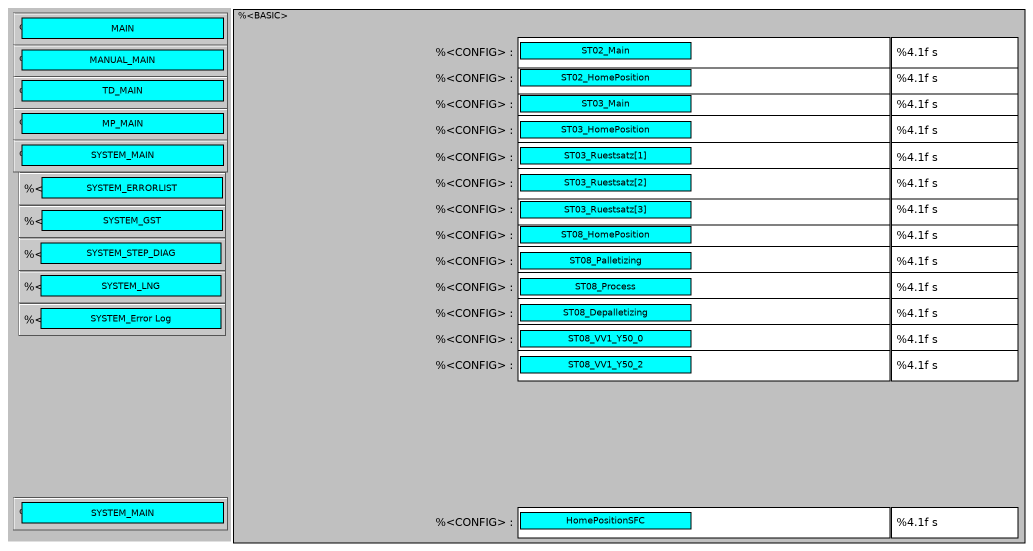
[picture p142: SYSTEM_STEP_DIAG (HMI screen)]
rectangle at (228,115)-(1020,649): text "%<BASIC>"; shows 'Prozess-Schrittketten'
embedded screen at (3,114)-(226,647): M0003_System
embedded screen at (282,195)-(1013,226): ZLIB_SFC_STATE
embedded screen at (282,221)-(1013,252): ZLIB_SFC_STATE
embedded screen at (282,326)-(1013,357): ZLIB_SFC_STATE
embedded screen at (282,352)-(1013,383): ZLIB_SFC_STATE
embedded screen at (282,378)-(1013,409): ZLIB_SFC_STATE
embedded screen at (282,404)-(1013,435): ZLIB_SFC_STATE
embedded screen at (282,430)-(1013,461): ZLIB_SFC_STATE
embedded screen at (282,456)-(1013,487): ZLIB_SFC_STATE
embedded screen at (282,300)-(1013,331): ZLIB_SFC_STATE; invisible if ST03_CallPRGs.ST03_Ruestsatz[3].b_activ
embedded screen at (282,613)-(1013,644): ZLIB_SFC_STATE
embedded screen at (282,169)-(1013,200): ZLIB_SFC_STATE
embedded screen at (282,143)-(1013,174): ZLIB_SFC_STATE
rectangle at (515,148)-(686,165): text "ST02_Main"; invisible if TRUE
rectangle at (515,175)-(686,192): text "ST02_HomePosition"; invisible if TRUE
rectangle at (515,201)-(686,218): text "ST03_Main"; invisible if TRUE
rectangle at (515,227)-(686,244): text "ST03_HomePosition"; invisible if TRUE
rectangle at (515,332)-(686,349): text "ST08_HomePosition"; invisible if TRUE
rectangle at (515,358)-(686,375): text "ST08_Palletizing"; invisible if TRUE
rectangle at (515,384)-(686,401): text "ST08_Process"; invisible if TRUE
rectangle at (515,410)-(686,427): text "ST08_Depalletizing"; invisible if TRUE
rectangle at (515,436)-(686,453): text "ST08_VV1_Y50_0"; invisible if TRUE
rectangle at (515,462)-(686,479): text "ST08_VV1_Y50_2"; invisible if TRUE
rectangle at (515,307)-(686,324): text "ST03_Ruestsatz[3]"; invisible if TRUE
rectangle at (515,618)-(686,635): text "HomePositionSFC"; invisible if TRUE
embedded screen at (282,248)-(1013,279): ZLIB_SFC_STATE; invisible if ST03_CallPRGs.ST03_Ruestsatz[1].b_activ
embedded screen at (282,274)-(1013,305): ZLIB_SFC_STATE; invisible if ST03_CallPRGs.ST03_Ruestsatz[2].b_activ
rectangle at (515,253)-(686,270): text "ST03_Ruestsatz[1]"; invisible if TRUE
rectangle at (515,280)-(686,297): text "ST03_Ruestsatz[2]"; invisible if TRUE
*)

(* Visualisation SIGNS_AXIS
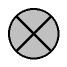
ellipse at (0,0)-(51,51): alarm colour if $Object$.on
polyline at (8,8)-(43,43): angle $Object$.sPos.lr_Mod /4
polyline at (8,8)-(43,43): angle $Object$.sPos.lr_Mod /4
*)

(* Visualisation ZLIB_7211_ACHSE
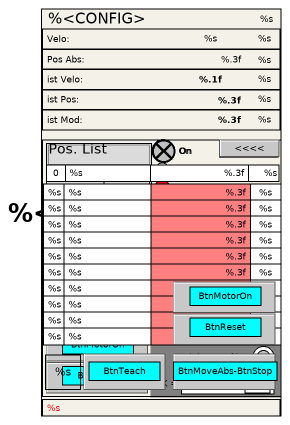
embedded screen at (0,0)-(241,408): ZLIB_7211_Control
embedded screen at (1,131)-(240,388): ZLIB_7211_ACHSE_Poslist; invisible if NOT $Object$.sVisuAxis.Poslist
*)

(* Visualisation ZLIB_7211_ACHSE_POSLIST
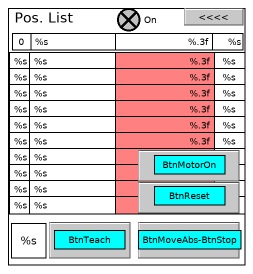
rectangle at (0,0)-(237,257): text "Pos. List"
rectangle at (22,25)-(108,42): text "%s"; shows $Offset$.Description; alarm colour if $Object$.sVisuAxis.PosNr = 0; editable; dynamic style ModeSelect.Mode>10
rectangle at (107,25)-(205,42): text "%.3f"; shows $Offset$.Pos; alarm colour if $Object$.sVisuAxis.PosNr = 0; editable; dynamic style ModeSelect.Mode>10 OR $Object$.On
rectangle at (204,25)-(235,42): text "%s"; shows $Object$.sVisuAxis.Einheit_pos; alarm colour if $Object$.sVisuAxis.PosNr = 0
embedded screen at (1,44)-(237,63): ZLIB_7211_ACHSE_POSLIST_LINE
embedded screen at (1,60)-(237,79): ZLIB_7211_ACHSE_POSLIST_LINE
embedded screen at (1,76)-(237,95): ZLIB_7211_ACHSE_POSLIST_LINE
embedded screen at (1,92)-(237,111): ZLIB_7211_ACHSE_POSLIST_LINE
rectangle at (3,215)-(38,250): text "%s"; shows $Object$.sVisuAxis.PosNr; editable 1..NO_OF_POS_AXIS
embedded screen at (1,108)-(237,127): ZLIB_7211_ACHSE_POSLIST_LINE
embedded screen at (1,124)-(237,143): ZLIB_7211_ACHSE_POSLIST_LINE
embedded screen at (1,140)-(237,159): ZLIB_7211_ACHSE_POSLIST_LINE
embedded screen at (1,156)-(237,175): ZLIB_7211_ACHSE_POSLIST_LINE
embedded screen at (1,172)-(237,191): ZLIB_7211_ACHSE_POSLIST_LINE
embedded screen at (1,188)-(237,207): ZLIB_7211_ACHSE_POSLIST_LINE
rectangle at (4,25)-(23,42): text "0"; invisible if TRUE; alarm colour if $Object$.sVisuAxis.PosNr = 0
button at (41,214)-(122,250): text "%<BTN>"; shows $Object$.sVisuAxis.BtnTeach.Text; invisible if NOT $Object$.sVisuAxis.BtnTeach.Visible; taps $Object$.sVisuAxis.BtnTeach.Pressed; dynamic style $Object$.sVisuAxis.BtnTeach.TextColor, $Object$.sVisuAxis.BtnTeach.BackgroundColor, $Object$.sVisuAxis.BtnTeach.BackgroundColor, NOT $Object$.sVisuAxis.BtnTeach.Enable
button at (130,214)-(231,250): text "%<BTN>"; shows $Object$.sVisuAxis.BtnMoveAbs.Text; invisible if NOT $Object$.sVisuAxis.BtnMoveAbs.Visible; taps $Object$.sVisuAxis.BtnMoveAbs.Pressed; dynamic style $Object$.sVisuAxis.BtnMoveAbs.TextColor, $Object$.sVisuAxis.BtnMoveAbs.BackgroundColor, $Object$.sVisuAxis.BtnMoveAbs.BackgroundColor, NOT $Object$.sVisuAxis.BtnMoveAbs.Enable
button at (130,214)-(231,250): text "%<BTN>"; shows $Object$.sVisuAxis.BtnStop.Text; invisible if NOT $Object$.sVisuAxis.BtnStop.Visible; taps $Object$.sVisuAxis.BtnStop.Pressed; dynamic style $Object$.sVisuAxis.BtnStop.TextColor, $Object$.sVisuAxis.BtnStop.BackgroundColor, $Object$.sVisuAxis.BtnStop.BackgroundColor, NOT $Object$.sVisuAxis.BtnStop.Enable
rectangle at (130,222)-(233,241): text "BtnMoveAbs-BtnStop"; invisible if TRUE
rectangle at (46,222)-(117,241): text "BtnTeach"; invisible if TRUE
rounded rectangle at (134,1)-(237,22): text "On"
embedded screen at (109,0)-(132,23): SIGNS_Axis
button at (176,0)-(235,17): text "<<<<"; toggles $Object$.sVisuAxis.Poslist; dynamic style Color.lightgrey
button at (130,142)-(231,173): text "%<BTN>"; shows $Object$.sVisuAxis.BtnMotorOn.Text; invisible if NOT $Object$.sVisuAxis.BtnMotorOn.Visible; taps $Object$.sVisuAxis.BtnMotorOn.Pressed; dynamic style $Object$.sVisuAxis.BtnMotorOn.TextColor, $Object$.sVisuAxis.BtnMotorOn.BackgroundColor, $Object$.sVisuAxis.BtnMotorOn.BackgroundColor, NOT $Object$.sVisuAxis.BtnMotorOn.Enable
button at (130,174)-(231,205): text "%<BTN>"; shows $Object$.sVisuAxis.BtnReset.Text; invisible if NOT $Object$.sVisuAxis.BtnReset.Visible; taps $Object$.sVisuAxis.BtnReset.Pressed; dynamic style $Object$.sVisuAxis.BtnReset.TextColor, $Object$.sVisuAxis.BtnReset.BackgroundColor, $Object$.sVisuAxis.BtnReset.BackgroundColor, NOT $Object$.sVisuAxis.BtnReset.Enable
rectangle at (146,147)-(217,166): text "BtnMotorOn"; invisible if TRUE
rectangle at (146,178)-(217,197): text "BtnReset"; invisible if TRUE
*)

(* Visualisation ZLIB_7211_ACHSE_POSLIST_LINE
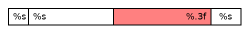
rectangle at (0,0)-(21,17): text "%s"; shows $Nr$; invisible if $Nr$ > NO_OF_POS_AXIS; alarm colour if $Object$.sVisuAxis.PosNr = $Nr$; toggles $Object$.sVisuAxis.b_Pos_nr[$Nr$]
rectangle at (105,0)-(203,17): text "%.3f"; shows $Poslist$[$Nr$].Pos; invisible if $Nr$ > NO_OF_POS_AXIS; alarm colour if $Object$.sVisuAxis.PosNr = $Nr$; editable $Object$.sConfig.SW_Limit_min..$Object$.sConfig.SW_Limit_max; dynamic style ModeSelect.Mode>10
rectangle at (202,0)-(233,17): text "%s"; shows $Object$.sVisuAxis.Einheit_pos; invisible if $Nr$ > NO_OF_POS_AXIS; alarm colour if $Object$.sVisuAxis.PosNr = $Nr$; toggles $Object$.sVisuAxis.b_Pos_nr[$Nr$]
rectangle at (20,0)-(106,17): text "%s"; shows $Poslist$[$Nr$].Description; invisible if $Nr$ > NO_OF_POS_AXIS; alarm colour if $Object$.sVisuAxis.PosNr = $Nr$; editable; dynamic style ModeSelect.Mode>10
rectangle at (105,0)-(203,17): text "%.3f"; shows $Poslist$[$Nr$].Pos; invisible if ($Poslist$[$Nr$].Pos >= $Object$.sConfig.SW_Limit_min AND $Poslist$[$Nr$].Pos <= $Object$.sConfig.SW_Limit_max)  OR $Nr$ > NO_OF_POS_AXIS; alarm colour if $Object$.sVisuAxis.PosNr = $Nr$; editable $Object$.sConfig.SW_Limit_min..$Object$.sConfig.SW_Limit_max; dynamic style ModeSelect.Mode>10
rectangle at (20,1)-(106,18): invisible if $Nr$ > NO_OF_POS_AXIS; toggles $Object$.sVisuAxis.b_Pos_nr[$Nr$]
*)

(* Visualisation ZLIB_7211_CONTROL
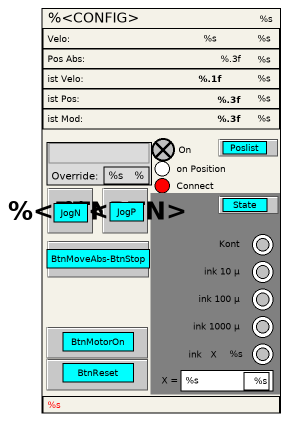
rectangle at (0,0)-(239,405): text "%<CONFIG>"; shows $Object$.sConfig.InstName
rectangle at (1,80)-(238,101): text "ist Pos:"; shows $Object$.sctrl.in.Position
rectangle at (1,100)-(238,121): text "ist Mod:"; shows $Object$.sPos.lr_Mod; invisible if NOT $Object$.sConfig.Modulo
rounded rectangle at (130,0)-(236,21): text "%s"; shows $Object$.sConfig.InstName
rectangle at (1,388)-(238,405): text "%s"; shows $Object$.LaufschriftObj.Display; invisible if $Object$.LaufschriftObj.Display=''
rectangle at (1,20)-(238,41): text "Velo:"; shows $Object$.Vorgabe_Velo; editable - $Object$.sVelo.maxRpm..$Object$.sVelo.maxRpm; dynamic style  ModeSelect.Mode>10
rectangle at (1,60)-(238,81): text "ist Velo:"; shows $Object$.sVelo.ist; alarm colour if $Object$.sVelo.dif >150 AND $Object$.on
rounded rectangle at (135,131)-(238,152): text "On"
embedded screen at (110,130)-(133,153): SIGNS_Axis
rectangle at (1,40)-(238,61): text "Pos Abs:"; shows $Object$.Vorgabe_Pos_Abs; alarm colour if $Poslist$[$Object$.sVisuAxis.PosNr].Pos = $Object$.Vorgabe_Pos_Abs AND ModeSelect.Mode =10; editable $Object$.sConfig.SW_Limit_min..$Object$.sConfig.SW_Limit_max; dynamic style ModeSelect.Mode>10
rounded rectangle at (40,42)-(204,59): text "%.3f"; shows $Object$.Vorgabe_Pos_Abs; editable $Object$.sConfig.SW_Limit_min..$Object$.sConfig.SW_Limit_max; dynamic style  ModeSelect.Mode>10
rounded rectangle at (203,43)-(234,59): text "%s"; shows $Object$.sVisuAxis.Einheit_pos
rounded rectangle at (183,22)-(234,38): text "%s"; shows $Object$.sVisuAxis.Einheit_velo
rounded rectangle at (183,62)-(234,78): text "%s"; shows $Object$.sVisuAxis.Einheit_Velo
rounded rectangle at (203,82)-(234,98): text "%s"; shows $Object$.sVisuAxis.Einheit_Pos
rounded rectangle at (203,102)-(234,118): text "%s"; shows $Object$.sVisuAxis.Einheit_Pos; invisible if NOT $Object$.sConfig.Modulo
ellipse at (113,153)-(128,168): alarm colour if $Object$.On_Position
rounded rectangle at (133,150)-(240,171): text "on Position"
rounded rectangle at (8,22)-(180,38): text "%s"; shows $Object$.Vorgabe_Velo; editable 0..$Object$.sVelo.maxRpm; dynamic style  ModeSelect.Mode>10
ellipse at (113,170)-(128,185): alarm colour if $Object$.Connect
rounded rectangle at (133,167)-(240,188): text "Connect"
button at (177,131)-(236,148): text "Pos. List"; invisible if $Poslist_unsichtbar$; toggles $Object$.sVisuAxis.Poslist; dynamic style Color.lightgrey
embedded screen at (5,134)-(110,177): ZLIB_OVERRIDE; dynamic style $Object$.sVisuAxis.Poslist
rectangle at (181,133)-(225,146): text "Poslist"; invisible if TRUE
other_LINEWIDTH at (109,185)-(238,386): invisible if $Object$.sVisuAxis.Control
embedded screen at (109,185)-(238,386): ZLIB_7211_OPT; invisible if NOT $Object$.sVisuAxis.Control
button at (6,180)-(51,225): text "%<BTN>"; shows $Object$.sVisuAxis.BtnJogm.Text; invisible if NOT $Object$.sVisuAxis.BtnJogM.Visible; taps $Object$.sVisuAxis.BtnJogM.Pressed; dynamic style $Object$.sVisuAxis.BtnJogM.TextColor, $Object$.sVisuAxis.BtnJogM.BackgroundColor, $Object$.sVisuAxis.BtnJogM.BackgroundColor, NOT $Object$.sVisuAxis.BtnJogM.Enable
button at (61,180)-(106,225): text "%<BTN>"; shows $Object$.sVisuAxis.BtnJogP.Text; invisible if NOT $Object$.sVisuAxis.BtnJogP.Visible; taps $Object$.sVisuAxis.BtnJogP.Pressed; dynamic style $Object$.sVisuAxis.BtnJogP.TextColor, $Object$.sVisuAxis.BtnJogP.BackgroundColor, $Object$.sVisuAxis.BtnJogP.BackgroundColor, NOT $Object$.sVisuAxis.BtnJogP.Enable
rectangle at (68,194)-(102,213): text "JogP"; invisible if TRUE
rectangle at (12,195)-(46,214): text "JogN"; invisible if TRUE
button at (5,319)-(106,350): text "%<BTN>"; shows $Object$.sVisuAxis.BtnMotorOn.Text; invisible if NOT $Object$.sVisuAxis.BtnMotorOn.Visible; taps $Object$.sVisuAxis.BtnMotorOn.Pressed; dynamic style $Object$.sVisuAxis.BtnMotorOn.TextColor, $Object$.sVisuAxis.BtnMotorOn.BackgroundColor, $Object$.sVisuAxis.BtnMotorOn.BackgroundColor, NOT $Object$.sVisuAxis.BtnMotorOn.Enable
button at (5,351)-(106,382): text "%<BTN>"; shows $Object$.sVisuAxis.BtnReset.Text; invisible if NOT $Object$.sVisuAxis.BtnReset.Visible; taps $Object$.sVisuAxis.BtnReset.Pressed; dynamic style $Object$.sVisuAxis.BtnReset.TextColor, $Object$.sVisuAxis.BtnReset.BackgroundColor, $Object$.sVisuAxis.BtnReset.BackgroundColor, NOT $Object$.sVisuAxis.BtnReset.Enable
rectangle at (21,324)-(92,343): text "BtnMotorOn"; invisible if TRUE
rectangle at (21,355)-(92,374): text "BtnReset"; invisible if TRUE
rectangle at (84,60)-(185,81): text "%.1f"; shows $Object$.sVelo.ist
rectangle at (53,81)-(204,102): text "%.3f"; shows $Object$.sctrl.in.Position
rectangle at (53,100)-(204,121): text "%.3f"; shows $Object$.sPos.lr_Mod; invisible if NOT $Object$.sConfig.Modulo
button at (6,233)-(107,269): text "%<BTN>"; shows $Object$.sVisuAxis.BtnMoveAbs.Text; invisible if NOT $Object$.sVisuAxis.BtnMoveAbs.Visible; taps $Object$.sVisuAxis.BtnMoveAbs.Pressed; dynamic style $Object$.sVisuAxis.BtnMoveAbs.TextColor, $Object$.sVisuAxis.BtnMoveAbs.BackgroundColor, $Object$.sVisuAxis.BtnMoveAbs.BackgroundColor, NOT $Object$.sVisuAxis.BtnMoveAbs.Enable
button at (6,233)-(107,269): text "%<BTN>"; shows $Object$.sVisuAxis.BtnStop.Text; invisible if NOT $Object$.sVisuAxis.BtnStop.Visible; taps $Object$.sVisuAxis.BtnStop.Pressed; dynamic style $Object$.sVisuAxis.BtnStop.TextColor, $Object$.sVisuAxis.BtnStop.BackgroundColor, $Object$.sVisuAxis.BtnStop.BackgroundColor, NOT $Object$.sVisuAxis.BtnStop.Enable
rectangle at (5,241)-(108,260): text "BtnMoveAbs-BtnStop"; invisible if TRUE
1 more shapes without text or variables
*)

(* Visualisation ZLIB_7211_OPT
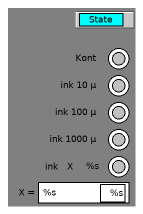
rectangle at (0,0)-(127,198): invisible if TRUE
ellipse at (100,40)-(121,61): alarm colour if $Object$.sVisuAxis.b_kont; toggles $Object$.sVisuAxis.b_kont; dynamic style  ModeSelect.Mode>10
ellipse at (104,44)-(117,57): alarm colour if $Object$.sVisuAxis.b_kont; toggles $Object$.sVisuAxis.b_kont; dynamic style  ModeSelect.Mode>10
ellipse at (100,67)-(121,88): alarm colour if $Object$.sVisuAxis.b_ink_10; toggles $Object$.sVisuAxis.b_ink_10; dynamic style  ModeSelect.Mode>10
ellipse at (104,71)-(117,84): alarm colour if $Object$.sVisuAxis.b_ink_10; toggles $Object$.sVisuAxis.b_ink_10; dynamic style  ModeSelect.Mode>10
ellipse at (100,94)-(121,115): alarm colour if $Object$.sVisuAxis.b_ink_100; toggles $Object$.sVisuAxis.b_ink_100; dynamic style  ModeSelect.Mode>10
ellipse at (104,98)-(117,111): alarm colour if $Object$.sVisuAxis.b_ink_100; toggles $Object$.sVisuAxis.b_ink_100; dynamic style  ModeSelect.Mode>10
ellipse at (100,121)-(121,142): alarm colour if $Object$.sVisuAxis.b_ink_1000; toggles $Object$.sVisuAxis.b_ink_1000; dynamic style  ModeSelect.Mode>10
ellipse at (104,125)-(117,138): alarm colour if $Object$.sVisuAxis.b_ink_1000; toggles $Object$.sVisuAxis.b_ink_1000; dynamic style  ModeSelect.Mode>10
ellipse at (100,148)-(121,169): alarm colour if $Object$.sVisuAxis.b_ink_var; toggles $Object$.sVisuAxis.b_ink_var; dynamic style  ModeSelect.Mode>10
ellipse at (104,152)-(117,165): alarm colour if $Object$.sVisuAxis.b_ink_var; toggles $Object$.sVisuAxis.b_ink_var; dynamic style  ModeSelect.Mode>10
rectangle at (27,42)-(93,58): text "Kont"; toggles $Object$.sVisuAxis.b_kont
rectangle at (27,69)-(93,85): text "ink 10 µ"; toggles $Object$.sVisuAxis.b_ink_10
rectangle at (26,96)-(93,112): text "ink 100 µ"; toggles $Object$.sVisuAxis.b_ink_100
rectangle at (26,123)-(93,139): text "ink 1000 µ"; toggles $Object$.sVisuAxis.b_ink_1000
rectangle at (32,151)-(70,166): text "ink   X"; toggles $Object$.sVisuAxis.b_ink_var
rectangle at (75,150)-(94,166): text "%s"; shows $Object$.sVisuAxis.Einheit_Pos; toggles $Object$.sVisuAxis.b_ink_var
rectangle at (5,177)-(32,192): text "X ="; toggles $Object$.sVisuAxis.b_ink_var
rectangle at (30,174)-(121,195): text "%s"; shows $Object$.sVisuAxis.lr_ink_var; editable 0..; dynamic style  ModeSelect.Mode>10 OR $Object$.sVisuAxis.Poslist
rectangle at (92,176)-(117,194): text "%s"; shows $Object$.sVisuAxis.Einheit_Pos; dynamic style  ModeSelect.Mode>10 OR $Object$.sVisuAxis.Poslist
button at (67,3)-(126,20): text "<<<<"; toggles $Object$.sVisuAxis.Control; dynamic style Color.lightgrey
rectangle at (71,5)-(115,18): text "State"; invisible if TRUE
*)

(* Visualisation ZLIB_7211_STATE
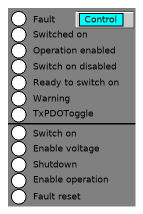
rectangle at (0,0)-(127,198): invisible if TRUE
ellipse at (3,67)-(18,82): alarm colour if $Object$.sCtrl.in.Ready_to_switch_on
rounded rectangle at (23,1)-(130,22): text "Fault"
ellipse at (3,19)-(18,34): alarm colour if $Object$.sCtrl.in.Switched_on
rounded rectangle at (23,16)-(130,37): text "Switched on"
ellipse at (3,35)-(18,50): alarm colour if $Object$.sCtrl.in.Operation_enabled
rounded rectangle at (23,32)-(130,53): text "Operation enabled"
ellipse at (3,3)-(18,18): alarm colour if $Object$.sCtrl.in.Fault
rounded rectangle at (23,64)-(130,85): text "Ready to switch on"
ellipse at (3,51)-(18,66): alarm colour if $Object$.sCtrl.in.Switch_on_disabled
rounded rectangle at (23,48)-(130,69): text "Switch on disabled"
ellipse at (3,83)-(18,98): alarm colour if $Object$.sCtrl.in.Warning
rounded rectangle at (23,80)-(130,101): text "Warning"
ellipse at (3,99)-(18,114): alarm colour if $Object$.sCtrl.in.TxPDOToggle
rounded rectangle at (23,95)-(130,116): text "TxPDOToggle"
ellipse at (3,117)-(18,132): alarm colour if $Object$.sCtrl.out.Switch_on
rounded rectangle at (23,115)-(130,136): text "Switch on"
ellipse at (3,133)-(18,148): alarm colour if $Object$.sCtrl.out.Enable_voltage
rounded rectangle at (23,130)-(130,151): text "Enable voltage"
ellipse at (3,149)-(18,164): alarm colour if $Object$.sCtrl.out.Shutdown
rounded rectangle at (23,146)-(130,167): text "Shutdown"
ellipse at (3,165)-(18,180): alarm colour if $Object$.sCtrl.out.Enable_operation
rounded rectangle at (23,161)-(130,182): text "Enable operation"
ellipse at (3,181)-(18,196): alarm colour if $Object$.sCtrl.out.Fault_reset
rounded rectangle at (23,178)-(130,199): text "Fault reset"
button at (67,3)-(126,20): text "Control"; invisible if ModeSelect.Mode > 10; toggles $Object$.sVisuAxis.Control; dynamic style Color.lightgrey
rectangle at (71,5)-(115,18): text "Control"; invisible if TRUE
1 more shapes without text or variables
*)

(* Visualisation DATA_HEADER
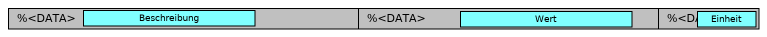
rectangle at (0,0)-(351,21): text "%<DATA>"; shows 'Description'
rectangle at (350,0)-(651,21): text "%<DATA>"; shows 'value'
rectangle at (650,0)-(751,21): text "%<DATA>"; shows 'unit'
rectangle at (75,2)-(247,18): text "Beschreibung"; invisible if TRUE
rectangle at (452,3)-(624,19): text "Wert"; invisible if TRUE
rectangle at (689,3)-(748,19): text "Einheit"; invisible if TRUE
*)

(* Visualisation DATA_LINE
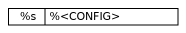
rectangle at (36,0)-(170,17): text "%<CONFIG>"; shows $Nr$; dynamic style ModeSelect.Mode<>MODE_MANUAL
rectangle at (0,0)-(37,17): text "%s"; shows '$Nr$'; dynamic style ModeSelect.Mode<>MODE_MANUAL
*)

(* Visualisation DATA_LINE_B
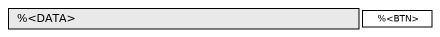
rectangle at (0,0)-(351,21): text "%<DATA>"; shows $Objekt$.Description; dynamic style NOT gst_datensatz.ST_MP.Inbetriebnahme.b
rounded rectangle at (354,2)-(424,19): text "%<BTN>"; shows 'on/off'; alarm colour if $Objekt$.b; toggles $Objekt$.b; dynamic style $deaktivieren$
rounded rectangle at (354,2)-(424,19): text "%<BTN>"; shows 'on/off'; invisible if $deaktivieren$; alarm colour if $Objekt$.b; toggles $Objekt$.b; dynamic style $deaktivieren$
*)

(* Visualisation DATA_LINE_BYTE
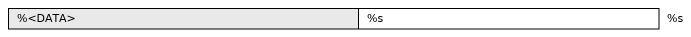
rectangle at (0,0)-(351,21): text "%<DATA>"; shows $Objekt$.Description; dynamic style NOT gst_datensatz.ST_MP.Inbetriebnahme.b
rectangle at (350,0)-(651,21): text "%s"; shows $Objekt$.BYT; editable 0..255; dynamic style $deaktivieren$
rectangle at (650,0)-(751,21): text "%s"; shows $Objekt$.unit; tooltip $Objekt$.unit; editable; dynamic style TRUE
rectangle at (350,0)-(651,21): text "%s"; shows $Objekt$.BYT; invisible if $deaktivieren$; editable 0..255; dynamic style $deaktivieren$
*)

(* Visualisation DATA_LINE_I16
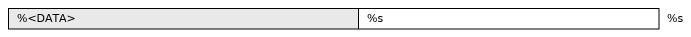
rectangle at (0,0)-(351,21): text "%<DATA>"; shows $Objekt$.Description; dynamic style NOT gst_datensatz.ST_MP.Inbetriebnahme.b
rectangle at (350,0)-(651,21): text "%s"; shows $Objekt$.i16; editable -32767..32767; dynamic style $deaktivieren$
rectangle at (650,0)-(751,21): text "%s"; shows $Objekt$.unit; invisible if $Objekt$.unit =''; tooltip $Objekt$.unit; editable; dynamic style TRUE
rectangle at (350,0)-(651,21): text "%s"; shows $Objekt$.i16; invisible if $deaktivieren$; editable -32767..32767; dynamic style $deaktivieren$
*)

(* Visualisation Data_LINE_i32
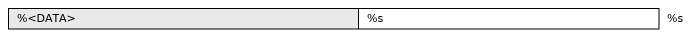
rectangle at (0,0)-(351,21): text "%<DATA>"; shows $Objekt$.Description; dynamic style NOT gst_datensatz.ST_MP.Inbetriebnahme.b
rectangle at (350,0)-(651,21): text "%s"; shows $Objekt$.i32; editable 0..; dynamic style $deaktivieren$
rectangle at (650,0)-(751,21): text "%s"; shows $Objekt$.unit; tooltip $Objekt$.unit; editable; dynamic style TRUE
rectangle at (350,0)-(651,21): text "%s"; shows $Objekt$.i32; invisible if $deaktivieren$; editable 0..; dynamic style $deaktivieren$
*)

(* Visualisation DATA_LINE_LR
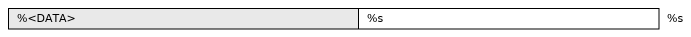
rectangle at (0,0)-(351,21): text "%<DATA>"; shows $Objekt$.Description; dynamic style NOT gst_datensatz.ST_MP.Inbetriebnahme.b
rectangle at (350,0)-(651,21): text "%s"; shows $Objekt$.lr; editable; dynamic style $deaktivieren$
rectangle at (650,0)-(751,21): text "%s"; shows $Objekt$.unit; tooltip $Objekt$.unit; editable; dynamic style TRUE
rectangle at (350,0)-(651,21): text "%s"; shows $Objekt$.lr; invisible if $deaktivieren$; editable; dynamic style $deaktivieren$
*)

(* Visualisation DATA_LINE_STR
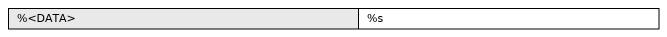
rectangle at (0,0)-(351,21): text "%<DATA>"; shows $Objekt$.Description; dynamic style NOT gst_datensatz.ST_MP.Inbetriebnahme.b
rectangle at (350,0)-(651,21): text "%s"; shows $Objekt$.str; editable; dynamic style $deaktivieren$
rectangle at (350,0)-(651,21): text "%s"; shows $Objekt$.str; invisible if $deaktivieren$; editable; dynamic style $deaktivieren$
*)

(* Visualisation Data_BOOL
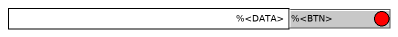
rectangle at (0,0)-(281,21): text "%<DATA>"; shows $Beschreibung$; invisible if $unsichtbar$
button at (281,1)-(382,20): text "%<BTN>"; shows 'On/Off'; invisible if $unsichtbar$; toggles $value$; dynamic style Color.lightgrey, Color.lightgrey, $deaktivieren$
button at (281,1)-(382,20): text "%<BTN>"; shows 'On/Off'; invisible if $unsichtbar$ OR $deaktivieren$; toggles $value$; dynamic style Color.lightgrey, Color.lightgrey, $deaktivieren$
ellipse at (366,3)-(381,18): invisible if $unsichtbar$; alarm colour if $value$
*)

(* Visualisation DATA_DEZIMAL
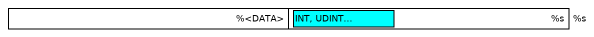
rectangle at (0,0)-(281,21): text "%<DATA>"; shows $Beschreibung$; invisible if $unsichtbar$; tooltip $Beschreibung$
rectangle at (280,0)-(561,21): text "%s"; shows $value$; invisible if $unsichtbar$; editable $MIN$..$MAX$; dynamic style $deaktivieren$
rectangle at (560,0)-(761,21): text "%s"; shows '$Einheit$'; invisible if $unsichtbar$; tooltip $Einheit$
rectangle at (280,0)-(561,21): text "%s"; shows $value$; invisible if $unsichtbar$ OR $deaktivieren$; editable $MIN$..$MAX$; dynamic style $deaktivieren$
rectangle at (285,2)-(386,19): text "INT, UDINT..."; invisible if TRUE
*)

(* Visualisation DATA_DEZIMAL_REAL
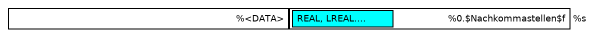
rectangle at (0,0)-(281,21): text "%<DATA>"; shows $Beschreibung$; invisible if $unsichtbar$; tooltip $Beschreibung$
rectangle at (280,0)-(561,21): text "%0.$Nachkommastellen$f"; shows $value$; invisible if $unsichtbar$; editable $MIN$..$MAX$; dynamic style $deaktivieren$
rectangle at (560,0)-(761,21): text "%s"; shows '$Einheit$'; invisible if $unsichtbar$; tooltip $Einheit$
rectangle at (281,0)-(562,21): text "%0.$Nachkommastellen$f"; shows $value$; invisible if $unsichtbar$ OR $deaktivieren$; editable $MIN$..$MAX$; dynamic style $deaktivieren$
rectangle at (284,2)-(385,19): text "REAL, LREAL...."; invisible if TRUE
*)

(* Visualisation DATA_HEADER_BEER
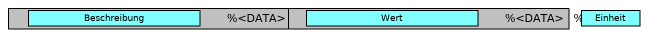
rectangle at (0,0)-(283,21): text "%<DATA>"; shows 'Description'
rectangle at (280,0)-(561,21): text "%<DATA>"; shows 'value'
rectangle at (560,0)-(641,21): text "%<DATA>"; shows 'unit'
rectangle at (20,2)-(192,18): text "Beschreibung"; invisible if TRUE
rectangle at (298,2)-(470,18): text "Wert"; invisible if TRUE
rectangle at (573,2)-(632,18): text "Einheit"; invisible if TRUE
*)

(* Visualisation DATA_STRING
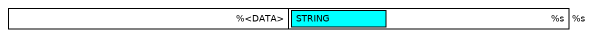
rectangle at (0,0)-(281,21): text "%<DATA>"; shows $Beschreibung$; invisible if $unsichtbar$
rectangle at (562,0)-(763,21): text "%s"; shows '$Einheit$'; invisible if $unsichtbar$; tooltip $Einheit$
rectangle at (280,0)-(561,21): text "%s"; shows $value$; invisible if $unsichtbar$; editable; dynamic style $deaktivieren$
rectangle at (280,0)-(561,21): text "%s"; shows $value$; invisible if $unsichtbar$ OR $deaktivieren$; editable; dynamic style $deaktivieren$
rectangle at (283,2)-(378,19): text "STRING"; invisible if TRUE
*)

(* Visualisation DIGIN
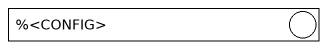
rounded rectangle at (1,1)-(280,32): text "%<CONFIG>"; shows '$Input$'
ellipse at (281,3)-(308,30): alarm colour if $Station$.$Input$; tooltip $Input$
1 more shapes without text or variables
*)

(* Visualisation DIGIN_red
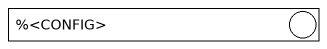
rounded rectangle at (1,1)-(280,32): text "%<CONFIG>"; shows '$Input$'
ellipse at (281,3)-(308,30): alarm colour if $Station$.$Input$; tooltip $Input$
1 more shapes without text or variables
*)

(* Visualisation DIGOUT_SMAL
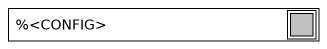
rectangle at (0,0)-(311,33): toggles $Station$.$Output$; dynamic style $OutputLocked$
rounded rectangle at (1,1)-(280,32): text "%<CONFIG>"; shows '$Output$'; toggles $Station$.$Output$; dynamic style $OutputLocked$
rounded rectangle at (279,2)-(308,31): alarm colour if $OutputLocked$; toggles $Station$.$Output$; dynamic style $OutputLocked$
rounded rectangle at (282,5)-(305,28): alarm colour if $Station$.$Output$; toggles $Station$.$Output$; tooltip $Output$; dynamic style $OutputLocked$
*)

(* Visualisation DIGOUT_TOUCH_SMAL
